// TIA Portal project "automated-assembly-cell" (V17)

(* hardware
DEVICE "S7-1200 station_1"  S7-1200 Station
   slot 0: "Rack_0"  S7-1200 Rack  Rack  V1.0
   slot 1: "PLC_Assembly_Cell"  CPU 1214C DC/DC/DC  6ES7 214-1AG40-0XB0  V4.5
DEVICE "HMI_Assembly_Cell"  KTP700 Basic PN
   slot 0: "HMI_Assembly_Cell"  KTP700 Basic PN  6AV2 123-2GB03-0AX0  17.0.0.0
   slot 1: "HMI_RT_2"  KTP700 Basic PN  6AV2 123-2GB03-0AX0  17.0.0.0
   slot 5: "HMI_Assembly_Cell.IE_CP_1"  PROFINET Interface  17.0.0.0
      slot 1: "PROFINET Interface_1"  PROFINET Interface
         slot 1: "Port_1"  Port
*)

// ===== PLC "PLC_Assembly_Cell"  CPU 1214C DC/DC/DC =====

VAR_GLOBAL   // PLC tag table "Input"
   "Start" AT %I0.0 : Bool;
   "Stop" AT %I0.1 : Bool;
   "Reset" AT %I0.2 : Bool;
   "EStop" AT %I0.3 : Bool;
   "Part_Sensor_in" AT %I0.4 : Bool;
   "Part_Sensor_Assembly" AT %I0.5 : Bool;
   "Part_Sensor_Out" AT %I0.6 : Bool;
   "Cylinder_Extended" AT %I0.7 : Bool;
   "Cylinder_Retracted" AT %I1.0 : Bool;
END_VAR

VAR_GLOBAL   // PLC tag table "Output"
   "Conveyor_Motor" AT %Q0.0 : Bool;
   "Cylinder_Extend" AT %Q0.1 : Bool;
   "Cylinder_Retract" AT %Q0.2 : Bool;
   "Green_lamp" AT %Q0.3 : Bool;
   "Red_Lamp" AT %Q0.4 : Bool;
   "Buzzer" AT %Q0.5 : Bool;
END_VAR

VAR_GLOBAL   // PLC tag table "Memories"
   "Machine_run" AT %M0.0 : Bool;
   "MAchine_Fault" AT %M0.1 : Bool;
   "Auto_Mode" AT %M0.2 : Bool;
   "Cycle_Active" AT %M0.3 : Bool;
   "Assembly_Complete" AT %M0.4 : Bool;
   "Satate" AT %MW2 : Int;
END_VAR

DATA_BLOCK "DB_Conveyor"   // DB1
{ S7_Optimized_Access := 'TRUE' }
AUTHOR : ING Miguel Angel Maldonado
VERSION : 0.1
// stored: InstanceOfName FB_Conveyor
"FB_Conveyor"
BEGIN
END_DATA_BLOCK

DATA_BLOCK "DB_Assembly"   // DB2
{ S7_Optimized_Access := 'TRUE' }
VERSION : 0.1
// stored: InstanceOfName FB_Assembly
"FB_Assembly"
BEGIN
END_DATA_BLOCK

FUNCTION_BLOCK "FB_Conveyor"   // FB1, LAD
{ S7_Optimized_Access := 'TRUE' }
AUTHOR : ING Miguel Angel Maldonado
VERSION : 0.1
   VAR_INPUT
      Eneable : Bool;
      Stop : Bool;
      Part_At_Assambly : Bool;
      Fault : Bool;
   END_VAR
   VAR_OUTPUT
      Motor : Bool;
   END_VAR
BEGIN

REGION Network 1
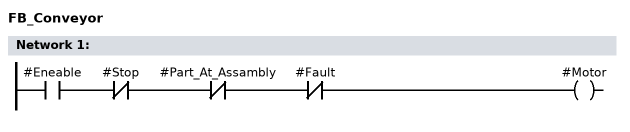
   RUNG wire#powerrail
      Contact( #Eneable )
      I_Contact( #Stop )
      I_Contact( #Part_At_Assambly )
      I_Contact( #Fault )
      Coil( #Motor )
   END_RUNG
   // the same network as SCL:
   #Motor := #Eneable AND NOT #Stop AND NOT #Part_At_Assambly AND NOT #Fault;
END_REGION
END_FUNCTION_BLOCK

FUNCTION_BLOCK "FB_Assembly"   // FB2, LAD
{ S7_Optimized_Access := 'TRUE' }
VERSION : 0.1
   VAR_INPUT
      Enable : Bool;   // Habilita el ciclo
      Start_Cycle : Bool;   // Solicita comenzar un ciclo
      Part_At_Assembly : Bool;   // Pieza Posicionada
      Cylinder_Extended : Bool;   // Confirmacion de Extension
      Cylinder_Retracted : Bool;   // Confirmacion de Retraccion
      Reset : Bool;   // Reinicia la secuencia
   END_VAR
   VAR_OUTPUT
      Cylinder_Extend : Bool;   // Orden Extender
      Cylinder_Retract : Bool;   // Orden de Retraer
      Assambly_Complete : Bool;   // Ciclo Terminado
      Assambly_Fault : Bool;   // Falla del Ciclo
   END_VAR
   VAR
      State : Int;
      Assambly_Timer : IEC_TIMER;
      Extend_Timeout : IEC_TIMER;
      Retract_Timeout : IEC_TIMER;
   END_VAR
BEGIN

REGION Network 1
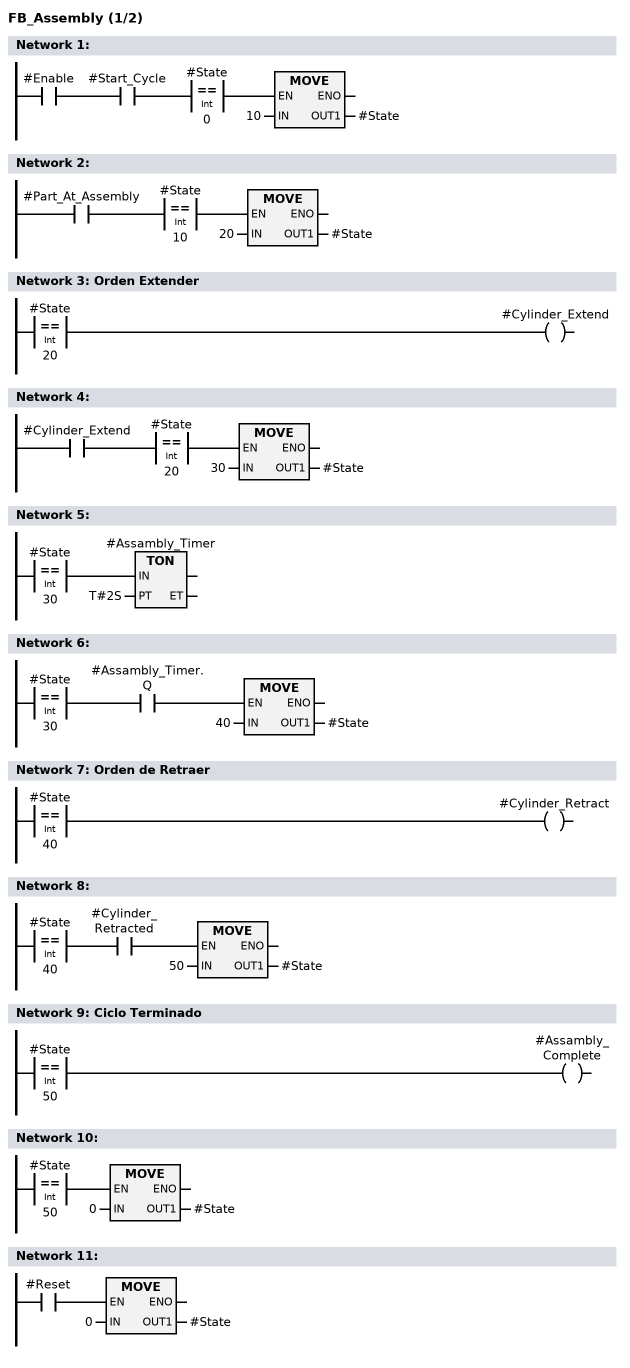
   RUNG wire#powerrail
      Contact( #Enable )
      Contact( #Start_Cycle )
      { S7_Templates := "SrcType := Int" } EQ_Contact(in1 := #State, in2 := 0)
      Move(in := 10, out1 => #State)
   END_RUNG
   // the same network as SCL:
   IF #Enable AND #Start_Cycle AND (#State = 0) THEN #State := 10; END_IF;
END_REGION

REGION Network 2
   RUNG wire#powerrail
      Contact( #Part_At_Assembly )
      { S7_Templates := "SrcType := Int" } EQ_Contact(in1 := #State, in2 := 10)
      Move(in := 20, out1 => #State)
   END_RUNG
   // the same network as SCL:
   IF #Part_At_Assembly AND (#State = 10) THEN #State := 20; END_IF;
END_REGION

REGION Network 3: Orden Extender
   RUNG wire#powerrail
      { S7_Templates := "SrcType := Int" } EQ_Contact(in1 := #State, in2 := 20)
      Coil( #Cylinder_Extend )
   END_RUNG
   // the same network as SCL:
   #Cylinder_Extend := #State = 20;
END_REGION

REGION Network 4
   RUNG wire#powerrail
      Contact( #Cylinder_Extend )
      { S7_Templates := "SrcType := Int" } EQ_Contact(in1 := #State, in2 := 20)
      Move(in := 30, out1 => #State)
   END_RUNG
   // the same network as SCL:
   IF #Cylinder_Extend AND (#State = 20) THEN #State := 30; END_IF;
END_REGION

REGION Network 5
   #Assambly_Timer.TON(IN := #State = 30, PT := T#2S);
END_REGION

REGION Network 6
   RUNG wire#powerrail
      { S7_Templates := "SrcType := Int" } EQ_Contact(in1 := #State, in2 := 30)
      Contact( #Assambly_Timer.Q )
      Move(in := 40, out1 => #State)
   END_RUNG
   // the same network as SCL:
   IF (#State = 30) AND #Assambly_Timer.Q THEN #State := 40; END_IF;
END_REGION

REGION Network 7: Orden de Retraer
   RUNG wire#powerrail
      { S7_Templates := "SrcType := Int" } EQ_Contact(in1 := #State, in2 := 40)
      Coil( #Cylinder_Retract )
   END_RUNG
   // the same network as SCL:
   #Cylinder_Retract := #State = 40;
END_REGION

REGION Network 8
   RUNG wire#powerrail
      { S7_Templates := "SrcType := Int" } EQ_Contact(in1 := #State, in2 := 40)
      Contact( #Cylinder_Retracted )
      Move(in := 50, out1 => #State)
   END_RUNG
   // the same network as SCL:
   IF (#State = 40) AND #Cylinder_Retracted THEN #State := 50; END_IF;
END_REGION

REGION Network 9: Ciclo Terminado
   RUNG wire#powerrail
      { S7_Templates := "SrcType := Int" } EQ_Contact(in1 := #State, in2 := 50)
      Coil( #Assambly_Complete )
   END_RUNG
   // the same network as SCL:
   #Assambly_Complete := #State = 50;
END_REGION

REGION Network 10
   RUNG wire#powerrail
      { S7_Templates := "SrcType := Int" } EQ_Contact(in1 := #State, in2 := 50)
      Move(in := 0, out1 => #State)
   END_RUNG
   // the same network as SCL:
   IF #State = 50 THEN #State := 0; END_IF;
END_REGION

REGION Network 11
   RUNG wire#powerrail
      Contact( #Reset )
      Move(in := 0, out1 => #State)
   END_RUNG
   // the same network as SCL:
   IF #Reset THEN #State := 0; END_IF;
END_REGION

REGION Network 12
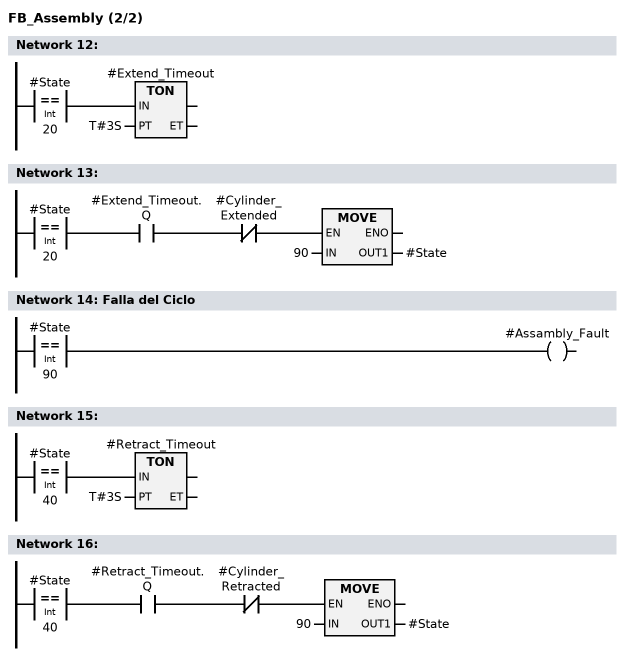
   #Extend_Timeout.TON(IN := #State = 20, PT := T#3S);
END_REGION

REGION Network 13
   RUNG wire#powerrail
      { S7_Templates := "SrcType := Int" } EQ_Contact(in1 := #State, in2 := 20)
      Contact( #Extend_Timeout.Q )
      I_Contact( #Cylinder_Extended )
      Move(in := 90, out1 => #State)
   END_RUNG
   // the same network as SCL:
   IF (#State = 20) AND #Extend_Timeout.Q AND NOT #Cylinder_Extended THEN #State := 90; END_IF;
END_REGION

REGION Network 14: Falla del Ciclo
   RUNG wire#powerrail
      { S7_Templates := "SrcType := Int" } EQ_Contact(in1 := #State, in2 := 90)
      Coil( #Assambly_Fault )
   END_RUNG
   // the same network as SCL:
   #Assambly_Fault := #State = 90;
END_REGION

REGION Network 15
   #Retract_Timeout.TON(IN := #State = 40, PT := T#3S);
END_REGION

REGION Network 16
   RUNG wire#powerrail
      { S7_Templates := "SrcType := Int" } EQ_Contact(in1 := #State, in2 := 40)
      Contact( #Retract_Timeout.Q )
      I_Contact( #Cylinder_Retracted )
      Move(in := 90, out1 => #State)
   END_RUNG
   // the same network as SCL:
   IF (#State = 40) AND #Retract_Timeout.Q AND NOT #Cylinder_Retracted THEN #State := 90; END_IF;
END_REGION
END_FUNCTION_BLOCK

ORGANIZATION_BLOCK "Main"   // OB1, LAD, ProgramCycle
TITLE = "Main Program Sweep (Cycle)"
{ S7_Optimized_Access := 'TRUE' }
VERSION : 0.1
   VAR_INPUT
      Initial_Call : Bool;   // Initial call of this OB
      Remanence : Bool;   // =True, if remanent data are available
   END_VAR
BEGIN

REGION Network 1
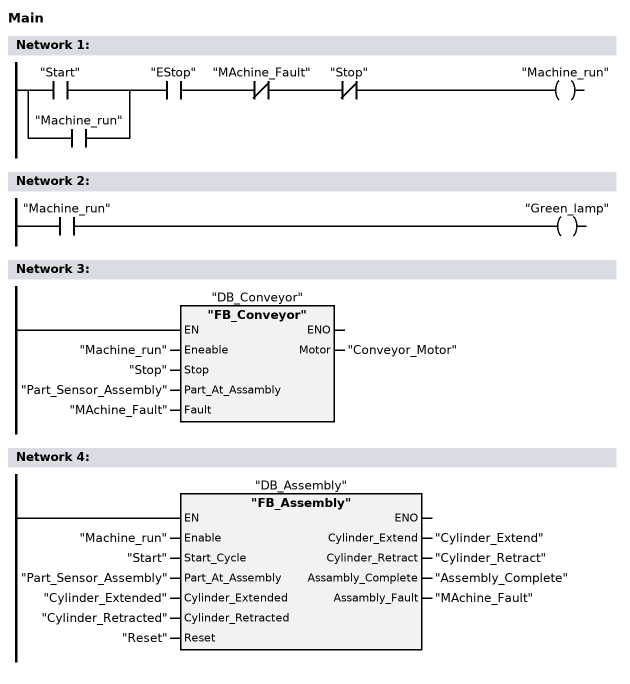
   RUNG wire#powerrail
      Contact( "Start" )
      wire#w1
      Contact( "EStop" )
      I_Contact( "MAchine_Fault" )
      I_Contact( "Stop" )
      Coil( "Machine_run" )
   END_RUNG
   RUNG wire#powerrail
      Contact( "Machine_run" )
   END_RUNG wire#w1
   // the same network as SCL:
   "Machine_run" := ("Start" OR "Machine_run") AND "EStop" AND NOT "MAchine_Fault" AND NOT "Stop";
END_REGION

REGION Network 2
   RUNG wire#powerrail
      Contact( "Machine_run" )
      Coil( "Green_lamp" )
   END_RUNG
   // the same network as SCL:
   "Green_lamp" := "Machine_run";
END_REGION

REGION Network 3
   RUNG wire#powerrail
      "DB_Conveyor"(Eneable := "Machine_run", Stop := "Stop", Part_At_Assambly := "Part_Sensor_Assembly", Fault := "MAchine_Fault", Motor => "Conveyor_Motor")
   END_RUNG
   // the same network as SCL:
   "DB_Conveyor"(Eneable := "Machine_run",   // "FB_Conveyor"
                 Stop := "Stop",
                 Part_At_Assambly := "Part_Sensor_Assembly",
                 Fault := "MAchine_Fault",
                 Motor => "Conveyor_Motor");
END_REGION

REGION Network 4
   RUNG wire#powerrail
      "DB_Assembly"(Enable := "Machine_run", Start_Cycle := "Start", Part_At_Assembly := "Part_Sensor_Assembly", Cylinder_Extended := "Cylinder_Extended", Cylinder_Retracted := "Cylinder_Retracted", Reset := "Reset", Cylinder_Extend => "Cylinder_Extend", Cylinder_Retract => "Cylinder_Retract", Assambly_Complete => "Assembly_Complete", Assambly_Fault => "MAchine_Fault")
   END_RUNG
   // the same network as SCL:
   "DB_Assembly"(Enable := "Machine_run",   // "FB_Assembly"
                 Start_Cycle := "Start",
                 Part_At_Assembly := "Part_Sensor_Assembly",
                 Cylinder_Extended := "Cylinder_Extended",
                 Cylinder_Retracted := "Cylinder_Retracted",
                 Reset := "Reset",
                 Cylinder_Extend => "Cylinder_Extend",
                 Cylinder_Retract => "Cylinder_Retract",
                 Assambly_Complete => "Assembly_Complete",
                 Assambly_Fault => "MAchine_Fault");
END_REGION
END_ORGANIZATION_BLOCK

(* ===== HMI "HMI_RT_2" =====
system functions are stored by id; their names below are inferred from use
connection "HMI_Connection_1": ETHERNET, SMART_S7_1200_OMS
connection "Connection_1": ETHERNET, SMART_S7_1200_OMS

HMI tags "Default tag table"
   "DB_Assembly_State" : Int = PLC DB_Assembly.State, 1 s
   "DB_Assembly_Cylinder_Retract" : Bool = PLC DB_Assembly.Cylinder_Retract, 1 s

HMI tags "PLC_Tags"
   "Start_PB" : Bool = PLC Start AT %I0.0, 1 s
   "Reset_PB" : Bool = PLC Reset AT %I0.2, 1 s
   "EStop_PB" : Bool = PLC EStop AT %I0.3, 1 s
   "Machine_Run" : Bool = PLC Machine_run AT %M0.0, 1 s
   "Machine_Fault" : Bool = PLC MAchine_Fault AT %M0.1, 1 s
   "Assembly_Complete" : Bool = PLC Assembly_Complete AT %M0.4, 1 s
   "Stop" : Bool = PLC Stop AT %I0.1, 1 s
   "Part_Sensor_Assembly" : Bool = PLC Part_Sensor_Assembly AT %I0.5, 1 s
   "Cylinder_Extended" : Bool = PLC Cylinder_Extended AT %I0.7, 1 s
   "Cylinder_Retracted" : Bool = PLC Cylinder_Retracted AT %I1.0, 1 s

screen "Main_Screen" 800x480
   Button "BTN_Start" at 70,416 size 126x56; TextOff 'START'
      on Press: SetBit("Start_PB")
      on Release: ResetBit("Start_PB")
   Button "BTN_Stop" at 320,416 size 126x56; TextOff 'STOP'
      on Release: ResetBit("Stop")
      on Press: SetBit("Stop")
   Button "BTN_RESET" at 570,416 size 126x56; TextOff 'RESET'
      on Release: ResetBit("Reset_PB")
      on Press: SetBit("Reset_PB")
   TextField "Text field_6" at 214,19 size 348x37; Text 'Automated Assambly Cell'
   TextField "Text field_7" at 150,100 size 93x34; Text 'STATUS'
   TextField "Text field_5" at 110,180 size 161x29; Text 'Part at Assembly'
   Circle "Lam_Part_at_assambly" at 50,180 size 32x32
      Appearance <- "Part_Sensor_Assembly"
   TextField "Text field_10" at 110,320 size 177x29; Text 'Cylinder Retracted'
   Circle "Lam_E-Stop_1" at 50,320 size 32x32
      Appearance <- "Cylinder_Retracted"
   TextField "Text field_9" at 110,250 size 174x29; Text 'Cylinder Extended'
   Circle "Lam_Machine_Fault_1" at 50,250 size 32x32
      Appearance <- "Cylinder_Extended"
   Group "Group" at 500,100 size 236x282
   TextField "Text field_8" at 500,100 size 110x34; Text 'MACHINE'
   TextField "Text field_1" at 550,180 size 45x29; Text 'RUN'
   Circle "Lam_Machine_Run" at 500,180 size 32x32
      Appearance <- "Machine_Run"
   TextField "Text field_2" at 550,240 size 50x29; Text 'Fault'
   Circle "Lam_Machine_Fault" at 500,240 size 32x32
      Appearance <- "Machine_Fault"
   TextField "Text field_3" at 550,350 size 66x29; Text 'E-Stop'
   Circle "Lam_E-Stop" at 500,350 size 32x32
      Appearance <- "EStop_PB"
   Circle "Lam_Assamby_Complete" at 500,300 size 32x32
      Appearance <- "Assembly_Complete"
   TextField "Text field_4" at 550,300 size 186x29; Text 'Assambly Complete'
*)